// TIA Portal V20 export
// export: Created 2026-09-01T12:42:15.710481Z, ExportSetting WithDefaults, DisplayName Totally Integrated Automation Portal, DisplayVersion V20 Update 5, DisplayName TIA Portal Openness, DisplayVersion V20 Update 4, DisplayName TIA Portal Version Control Interface, DisplayVersion V20 Update 5, DisplayName SINAMICS Startdrive Advanced, DisplayVersion V20, DisplayName SINAMICS DCC, DisplayVersion V20, DisplayName SINAMICS Startdrive G130, G150, S120, S150, SINAMICS MV, G220, S200, S210, DisplayVersion V20, DisplayName SINAMICS Startdrive G110M, G120, G120C, G120D, G120P, G115D, DisplayVersion V20, DisplayName STEP 7 Professional, DisplayVersion V20 Update 5, DisplayName STEP 7 Safety, DisplayVersion V20 Update 2, DisplayName WinCC Basic/Comfort/Advanced, DisplayVersion V20 Update 5, DisplayName WinCC Unified, DisplayVersion V20 Update 5
FUNCTION_BLOCK "FB_HopperBlockageMonitor"   // FB50, LAD
TITLE = Hopper-Blockage Monitor
{ S7_Optimized_Access := 'TRUE' }
VERSION : 0.1
// Supervises the shredder hopper high-level sensor: raises a latched hopper-blockage alarm (and a stop/inhibit demand) when the hopper stays (debounced-)high for a cumulative threshold of time while the plant is running, i.e. the shredder/pusher is not clearing it (S6 request #1, REQ-HBA-001..007). Purely supervisory - it commands no motion and writes no shared tag; the alarm and the stop demand are exposed on its own IO interface and wired to annunciation / the actual stop at a separate integration step (Q-HBA-05). Cumulative timing is pause-and-resume (NEW-HBA-01): losing PlantRunning freezes the elapsed and resumes, so 60 s of blockage need not be contiguous. Built from a plain TON, never TONR (C-406), plus a banked up-accumulator compared against the threshold (see NETWORK 3-4). The alarm latch lives in the RETAIN interface and deliberately survives a power cycle (C-124 carve-out, NEW-HBA-04) - like the sequencer's DischargeConveyorTimeoutFault, a blockage needing a human still needs FaultReset after a restart; all transient timing state is non-retentive and self-clears at startup (NEW-HBA-06, no OB100 edit). Tunables BlockedTimeThreshold (T#60S) and ClearDebounceTime (T#2S) are this instance's own settings (C-307), not shared DB members.
// stored: AutoNumber true, IsIECCheckEnabled false, IsRetainMemResEnabled false, MemoryReserve 100, SetENOAutomatically false, UDAEnableTagReadback false
   VAR RETAIN
      IO { S7_SetPoint := 'True'} : "UDT_HopperBlockageIO";   // Caller interface (C-115). Inputs (HopperLevelHigh/PlantRunning/FaultReset) are written by FC_ControlMain at integration; outputs (HopperBlockedAlarm/HopperBlockedInhibit) are read there. The whole interface is RETAIN - immaterial for the re-driven inputs, deliberate for the two output latches (C-124 carve-out).
   END_VAR
   VAR
      HighQualified : Bool;   // Debounced blockage-present latch: set the instant the hopper reads high, held through momentary sensor clears (chatter), cleared only once the hopper has read clear continuously for ClearDebounceTime (Q-HBA-02). Transient (non-retentive).
      BlockActive : Bool;   // The persistence window accrues only while this is true: a qualified blockage AND the plant actually running (Q-HBA-04).
      BlockActiveMem : Bool;   // Previous-scan BlockActive, for the constructed falling-edge (C-404).
      PauseEdge : Bool;   // One-scan pulse when BlockActive falls (plant stop or genuine clear) - fires the T_SUB bank in NETWORK 4.
      FaultResetMem : Bool;   // Previous-scan copy of the operator FaultReset input; NETWORK 5 compares the two to find the moment it goes true. Transient (non-retentive).
      FaultResetEdge : Bool;   // One-scan pulse when FaultReset goes true - the operator acknowledgement that clears the alarm latch in NETWORK 5. A reset held on produces one pulse, not a continuous clear. Transient (non-retentive).
      AccumulatedElapsed : Time;   // Cumulative high-and-running elapsed banked across plant-stop pauses (NEW-HBA-01). Two writers (NETWORK 3) that can never fire in the same scan: back to T#0S on a confirmed clear, banked up by each just-ended segment's elapsed on a plant-stop pause. A FaultReset does not touch it (REQ-HBA-005). Transient (non-retentive); starts 0, so no first-scan trip.
      CumulativeElapsed : Time;   // Live total = AccumulatedElapsed + PersistenceTimer.ET (NETWORK 4), compared against BlockedTimeThreshold to trip the alarm. Single-writer, derived each scan.
      ZeroTime : Time;   // Constant zero (T#0S) source for the accumulator reset - TIA import rejects a bare Time literal as a MOVE operand, so the zero is held as an unwritten Time member (defaults to T#0S, never written). Non-retentive.
      ClearDebounceTimer { S7_SetPoint := 'True'} : TON_TIME;
      PersistenceTimer { S7_SetPoint := 'True'} : TON_TIME;
   END_VAR
BEGIN

REGION Network 1: Confirmed-Clear Debounce
   // Times the hopper reading NOT high. Its Q (hopper clear continuously for ClearDebounceTime) is the only thing that re-arms the blockage qualifier - a shorter blip is ignored (Q-HBA-02, debounced clear).
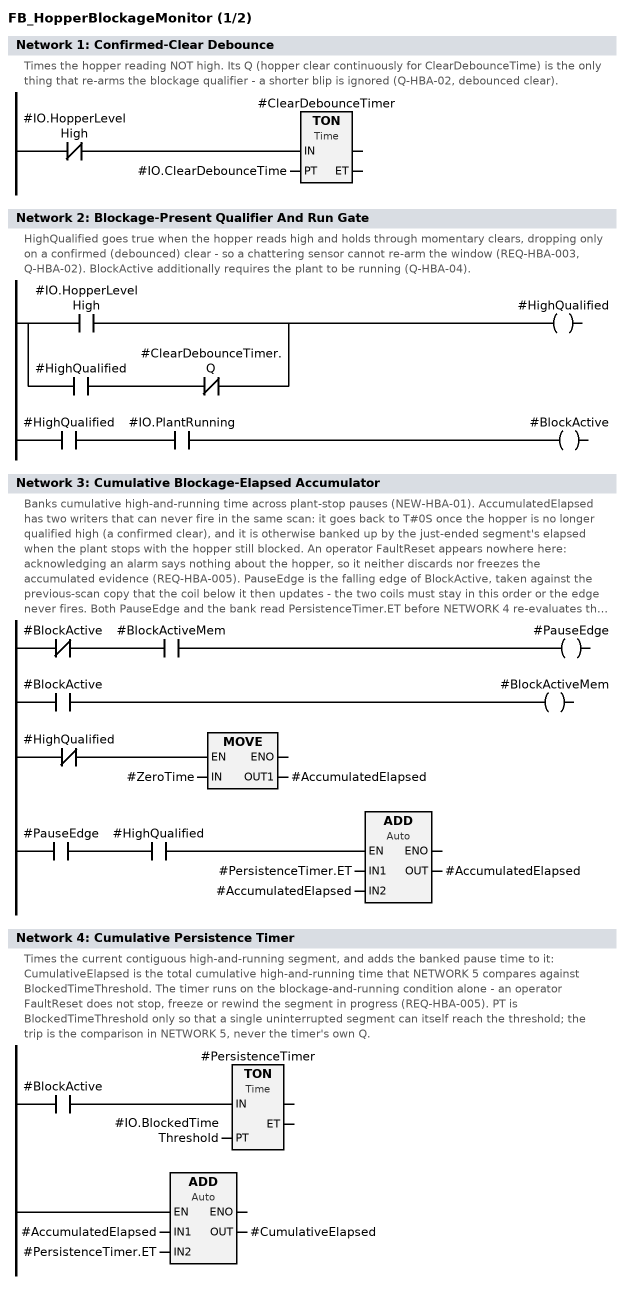
   RUNG wire#powerrail
      I_Contact( #IO.HopperLevelHigh )
      { S7_Templates := "time_type := Time" } #ClearDebounceTimer.TON(pt := #IO.ClearDebounceTime, et =>)
   END_RUNG
   // the same network as SCL:
   #ClearDebounceTimer(IN := NOT #IO.HopperLevelHigh, PT := #IO.ClearDebounceTime);   // TON
END_REGION

REGION Network 2: Blockage-Present Qualifier And Run Gate
   // HighQualified goes true when the hopper reads high and holds through momentary clears, dropping only on a confirmed (debounced) clear - so a chattering sensor cannot re-arm the window (REQ-HBA-003, Q-HBA-02). BlockActive additionally requires the plant to be running (Q-HBA-04).
   RUNG wire#powerrail
      Contact( #IO.HopperLevelHigh )
      wire#w1
      Coil( #HighQualified )
   END_RUNG
   RUNG wire#powerrail
      Contact( #HighQualified )
      I_Contact( #ClearDebounceTimer.Q )
   END_RUNG wire#w1
   RUNG wire#powerrail
      Contact( #HighQualified )
      Contact( #IO.PlantRunning )
      Coil( #BlockActive )
   END_RUNG
   // the same network as SCL:
   #HighQualified := #IO.HopperLevelHigh OR (#HighQualified AND NOT #ClearDebounceTimer.Q);
   #BlockActive := #HighQualified AND #IO.PlantRunning;
END_REGION

REGION Network 3: Cumulative Blockage-Elapsed Accumulator
   // Banks cumulative high-and-running time across plant-stop pauses (NEW-HBA-01). AccumulatedElapsed has two writers that can never fire in the same scan: it goes back to T#0S once the hopper is no longer qualified high (a confirmed clear), and it is otherwise banked up by the just-ended segment's elapsed when the plant stops with the hopper still blocked. An operator FaultReset appears nowhere here: acknowledging an alarm says nothing about the hopper, so it neither discards nor freezes the accumulated evidence (REQ-HBA-005). PauseEdge is the falling edge of BlockActive, taken against the previous-scan copy that the coil below it then updates - the two coils must stay in this order or the edge never fires. Both PauseEdge and the bank read PersistenceTimer.ET before NETWORK 4 re-evaluates the timer this scan, so the elapsed banked is the just-completed segment's, with no separate held-value register needed.
   RUNG wire#powerrail
      I_Contact( #BlockActive )
      Contact( #BlockActiveMem )
      Coil( #PauseEdge )
   END_RUNG
   RUNG wire#powerrail
      Contact( #BlockActive )
      Coil( #BlockActiveMem )
   END_RUNG
   RUNG wire#powerrail
      I_Contact( #HighQualified )
      Move(in := #ZeroTime, out1 => #AccumulatedElapsed)
   END_RUNG
   RUNG wire#powerrail
      Contact( #PauseEdge )
      Contact( #HighQualified )
      Add(in1 := #PersistenceTimer.ET, in2 := #AccumulatedElapsed, out => #AccumulatedElapsed)
   END_RUNG
   // the same network as SCL:
   #PauseEdge := NOT #BlockActive AND #BlockActiveMem;
   #BlockActiveMem := #BlockActive;
   IF NOT #HighQualified THEN #AccumulatedElapsed := #ZeroTime; END_IF;
   IF #PauseEdge AND #HighQualified THEN
       #AccumulatedElapsed := #PersistenceTimer.ET + #AccumulatedElapsed;
   END_IF;
END_REGION

REGION Network 4: Cumulative Persistence Timer
   // Times the current contiguous high-and-running segment, and adds the banked pause time to it: CumulativeElapsed is the total cumulative high-and-running time that NETWORK 5 compares against BlockedTimeThreshold. The timer runs on the blockage-and-running condition alone - an operator FaultReset does not stop, freeze or rewind the segment in progress (REQ-HBA-005). PT is BlockedTimeThreshold only so that a single uninterrupted segment can itself reach the threshold; the trip is the comparison in NETWORK 5, never the timer's own Q.
   RUNG wire#powerrail
      Contact( #BlockActive )
      { S7_Templates := "time_type := Time" } #PersistenceTimer.TON(pt := #IO.BlockedTimeThreshold, et =>)
   END_RUNG
   RUNG wire#powerrail
      Add(in1 := #AccumulatedElapsed, in2 := #PersistenceTimer.ET, out => #CumulativeElapsed)
   END_RUNG
   // the same network as SCL:
   #PersistenceTimer(IN := #BlockActive, PT := #IO.BlockedTimeThreshold);   // TON
   #CumulativeElapsed := #AccumulatedElapsed + #PersistenceTimer.ET;
END_REGION

REGION Network 5: Hopper-Blocked Alarm Latch (RETAIN - Survives Power Cycle)
   // Latches the hopper-blockage alarm when the cumulative high-and-running time reaches BlockedTimeThreshold, and holds it until an operator acknowledges. The acknowledgement is the moment FaultReset goes true, not the fact that it is true: a reset left on, wired on or stuck on clears the latch once and cannot hold the alarm off afterwards (REQ-HBA-005). Because the reset leaves the accumulated evidence alone, the latch re-evaluates on the very next scan against that same evidence - a hopper still blocked past the threshold re-alarms at once, whether or not the plant is running, while a hopper whose evidence has been discarded stays quiet. The reset pulse is taken against the previous-scan copy that the coil below it then updates - the two coils must stay in this order or the pulse never fires. The latch lives in the RETAIN interface and survives a power cycle: a blockage that needed a human still needs acknowledging after a restart, and the stop demand below stays asserted until it gets one.
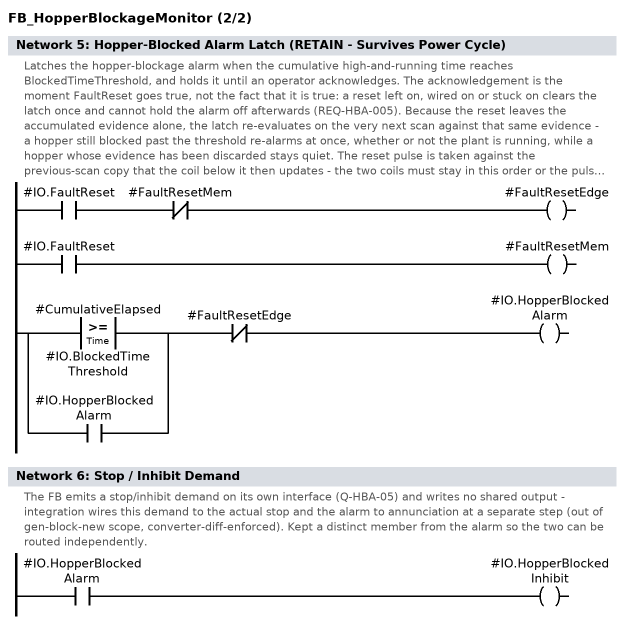
   RUNG wire#powerrail
      Contact( #IO.FaultReset )
      I_Contact( #FaultResetMem )
      Coil( #FaultResetEdge )
   END_RUNG
   RUNG wire#powerrail
      Contact( #IO.FaultReset )
      Coil( #FaultResetMem )
   END_RUNG
   RUNG wire#powerrail
      { S7_Templates := "SrcType := Time" } GE_Contact(in1 := #CumulativeElapsed, in2 := #IO.BlockedTimeThreshold)
      wire#w1
      I_Contact( #FaultResetEdge )
      Coil( #IO.HopperBlockedAlarm )
   END_RUNG
   RUNG wire#powerrail
      Contact( #IO.HopperBlockedAlarm )
   END_RUNG wire#w1
   // the same network as SCL:
   #FaultResetEdge := #IO.FaultReset AND NOT #FaultResetMem;
   #FaultResetMem := #IO.FaultReset;
   #IO.HopperBlockedAlarm := ((#CumulativeElapsed >= #IO.BlockedTimeThreshold) OR #IO.HopperBlockedAlarm) AND NOT #FaultResetEdge;
END_REGION

REGION Network 6: Stop / Inhibit Demand
   // The FB emits a stop/inhibit demand on its own interface (Q-HBA-05) and writes no shared output - integration wires this demand to the actual stop and the alarm to annunciation at a separate step (out of gen-block-new scope, converter-diff-enforced). Kept a distinct member from the alarm so the two can be routed independently.
   RUNG wire#powerrail
      Contact( #IO.HopperBlockedAlarm )
      Coil( #IO.HopperBlockedInhibit )
   END_RUNG
   // the same network as SCL:
   #IO.HopperBlockedInhibit := #IO.HopperBlockedAlarm;
END_REGION
END_FUNCTION_BLOCK
